// TIA Portal V19 export
DATA_BLOCK "PTrk_HMI"   // DB177
// stored: MemoryReserve 100
   VAR
      Button_Part_Recondition_Good : Struct
         Show : Bool;
         AllowControl : Bool;
         Pressed : Bool;
      END_STRUCT;
      Button_Part_Recondition_NG : Struct
         Show : Bool;
         AllowControl : Bool;
         Pressed : Bool;
      END_STRUCT;
   END_VAR
BEGIN
END_DATA_BLOCK
